FUNCTION_BLOCK PUBLIC FB_LampSetDirectDALIAdapter EXTENDS FB_Lamp
VAR
	fbLampSetDirectDALI		: FB_LampSetDirectDALI;
END_VAR

fbLampSetDirectDALI();

// Reduces the control value by 5 in the range of 10 to 254.
METHOD PUBLIC DimDown
IF (fbLampSetDirectDALI.nLightLevel >= 38.1) THEN
	fbLampSetDirectDALI.SetLightLevel(TO_USINT(fbLampSetDirectDALI.nLightLevel - 12.7));
END_IF
IF (_ipObserver <> 0) THEN
	_ipObserver.Update(TO_USINT(fbLampSetDirectDALI.nLightLevel * 100.0 / 254.0));
END_IF
END_METHOD

// Increments the control value by 5 in the range of 10 to 254.
METHOD PUBLIC DimUp
IF (fbLampSetDirectDALI.nLightLevel <= 241.3) THEN
	fbLampSetDirectDALI.SetLightLevel(TO_USINT(TO_LREAL(fbLampSetDirectDALI.nLightLevel) + 12.7));
END_IF
IF (_ipObserver <> 0) THEN
	_ipObserver.Update(TO_USINT(fbLampSetDirectDALI.nLightLevel * 100.0 / 254.0));
END_IF
END_METHOD

{attribute 'monitoring' := 'call'}
// Operating Time [s]
PROPERTY PUBLIC nOperatingTime : DINT
GET
nOperatingTime := fbLampSetDirectDALI.nOperatingTime;
END_GET
SET
fbLampSetDirectDALI.nOperatingTime := nOperatingTime;
END_SET
END_PROPERTY

// Sets the control value to 0.
METHOD PUBLIC Off
fbLampSetDirectDALI.SetLightLevel(0);
IF (_ipObserver <> 0) THEN
	_ipObserver.Update(TO_USINT(fbLampSetDirectDALI.nLightLevel * 100.0 / 254.0));
END_IF
END_METHOD

// Sets the control value to 254.
METHOD PUBLIC On
fbLampSetDirectDALI.SetLightLevel(254);
IF (_ipObserver <> 0) THEN
	_ipObserver.Update(TO_USINT(fbLampSetDirectDALI.nLightLevel * 100.0 / 254.0));
END_IF
END_METHOD

END_FUNCTION_BLOCK

(* stored: Version 1.1.0.1, ProductVersion 3.1.4024.12
   POU FB_LampSetDirectDALIAdapter: Id {06500677-1ca5-4f9c-bbca-0dcd0188c3d3}, SpecialFunc None
   Method DimDown: Id {7a075584-61ed-49e7-aa80-b192dd0ff064}
   Method DimUp: Id {85c48a51-31d1-4f15-b30f-dd92b0da00a7}
   Property nOperatingTime: Id {bac1895c-e0d1-4333-ab07-93d9798a159d}
   Get Get: Id {fa922e52-e840-4408-90d7-832311b52e47}
   Set Set: Id {58905beb-3546-486d-9cea-545eff8ce0c6}
   Method Off: Id {3106f1b1-a466-4aaf-bf7c-b90c0d8b4c22}
   Method On: Id {2094a9c9-f771-43f7-aa2d-1a5adb3e0e4e} *)
